Fanuc TP program (LS listing): CLSKP_G3.LS

/PROG  CLSKP_G3
/ATTR
OWNER		= MNEDITOR;
COMMENT		= "set skip cond g3";
PROG_SIZE	= 294;
CREATE		= DATE 08-10-17  TIME 22:35:34;
MODIFIED	= DATE 08-10-17  TIME 22:39:00;
FILE_NAME	= CLSKP_G2;
VERSION		= 0;
LINE_COUNT	= 6;
MEMORY_SIZE	= 642;
PROTECT		= READ_WRITE;
TCD:  STACK_SIZE	= 0,
      TASK_PRIORITY	= 50,
      TIME_SLICE	= 0,
      BUSY_LAMP_OFF	= 0,
      ABORT_REQUEST	= 0,
      PAUSE_REQUEST	= 0;
DEFAULT_GROUP	= *,*,*,*,*;
CONTROL_CODE	= 00000000 00000000;
/APPL
/APPL
/MN
   1:  !Program CLSKP_g3  ;
   2:   ;
   3:  SKIP CONDITION $MISC[3].$DSTB_EXCESS=1    ;
   4:  END ;
   5:   ;
   6:  !End of CLSKP_g3  ;
/POS
/END
